TYPE ST_HMI :
STRUCT
	stIn 	: ST_HMI_IN;
	stOut 	: ST_HMI_OUT;
END_STRUCT
END_TYPE

(* stored: Version 1.1.0.1, ProductVersion 3.1.4024.12
   DUT ST_HMI: Id {79311218-20e2-4d7b-b3ef-8a8affaeb9ab} *)
